Universal Robots PolyScope program: dlo_p0001.urp

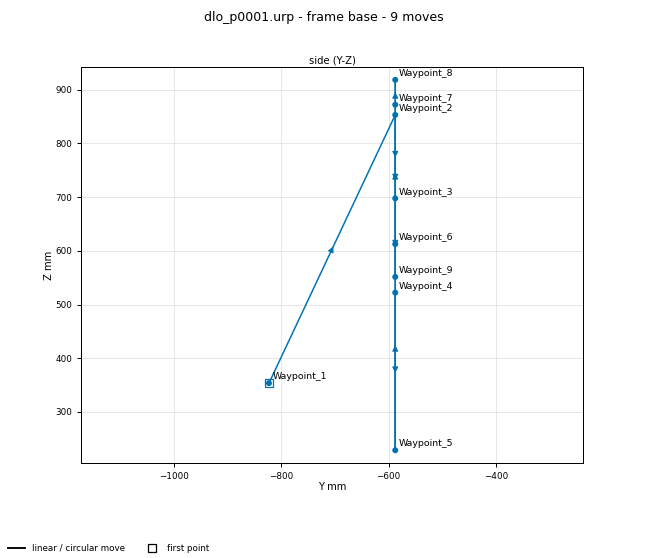
[picture p0: tool path of dlo_p0001.urp in frame base, 9 of 9 moves have a stored position in this frame; points joined in program order, loops and branches not executed]
Program dlo_p0001 (installation=dlo_01 directory=/programs/usbdisk/ur5e createdIn=5.11.4.108353 lastSavedIn=5.11.4.108353 robotSerialNumber=20205500325)
Calibrated DH parameters: a=[0.000117, -0.041718, -0.362867, 0.000002, -0.000002, 0]; d=[0.162762, 132.78066, -173.894578, 41.247059, 0.099793, 0.099638]; alpha=[1.568696, -0.003189, 0.003637, 1.569952, -1.569426, 0]; deltaTheta=[0, -1.472603, 7.364952, 0.390842, 0, 0]
Robot Program (runOnlyOnce=false)
  SetPayload (workpieceName=R2F85_payload)
  MoveJ speed 60 deg/s, acceleration 80 deg/s^2 (useActiveTCP=true) feature=Base
    Waypoint Waypoint_1: TCP in base x=10.232 y=-822.834 z=353.649 mm, rx=0.003 ry=-2.2345 rz=2.1939 rad; joints [76.813, -57.884, 100.068, -221.089, -77.331, -0.468] deg; TCP offset x=0 y=0 z=188 mm, rx=0 ry=0 rz=0 rad
    Popup Message (haltProgram=false message=Bring the DLO near the gripper for gripping, then continue inputType=Text)
    Wait Sleep waitTime=1
    URCap Gripper (Robotiq_Grippers, Robotiq Inc.) dataModel(position=100.0, force=100.0, speed=0.0, positionInDouble=100.0, forceInDouble=100.0, speedInDouble=0.0, slaveIds=[9], blocking=true)
  MoveL speed 250 mm/s, acceleration 1200 mm/s^2 (useActiveTCP=true) feature=Joint_6_name
    Waypoint Waypoint_2: TCP in base x=-0.89 y=-587.732 z=853.044 mm, rx=-0.0177 ry=-2.2261 rz=2.1975 rad; joints [64.46, -101.218, 74.368, -152.362, -65.292, -0.205] deg; feature pose in base x=-0.89 y=-587.732 z=853.044 mm, rx=-0.0177 ry=-2.2261 rz=2.1975 rad
    Waypoint Waypoint_3: TCP in base x=-0.933 y=-587.741 z=697.705 mm, rx=-0.0178 ry=-2.2261 rz=2.1974 rad; joints [64.497, -106.875, 102.164, -174.52, -65.377, -0.152] deg; feature pose in base x=-0.933 y=-587.741 z=697.705 mm, rx=-0.0178 ry=-2.2261 rz=2.1974 rad
    Waypoint Waypoint_4: TCP in base x=-0.931 y=-587.718 z=522.229 mm, rx=-0.0176 ry=-2.2259 rz=2.1975 rad; joints [64.51, -102.812, 125.433, -201.873, -65.499, -0.126] deg; feature pose in base x=-0.931 y=-587.718 z=522.229 mm, rx=-0.0176 ry=-2.2259 rz=2.1975 rad
    Waypoint Waypoint_5: TCP in base x=-0.913 y=-587.718 z=228.776 mm, rx=-0.0178 ry=-2.2261 rz=2.1974 rad; joints [64.493, -57.887, 141.707, -262.996, -65.801, -0.279] deg; feature pose in base x=-0.913 y=-587.718 z=228.776 mm, rx=-0.0178 ry=-2.2261 rz=2.1974 rad
    Waypoint Waypoint_6: TCP in base x=-0.894 y=-587.737 z=612.595 mm, rx=-0.0176 ry=-2.226 rz=2.1975 rad; joints [64.511, -106.524, 114.374, -187.092, -65.43, -0.134] deg; feature pose in base x=-0.894 y=-587.737 z=612.595 mm, rx=-0.0176 ry=-2.226 rz=2.1975 rad
    Waypoint Waypoint_7: TCP in base x=-0.868 y=-587.719 z=872.008 mm, rx=-0.0176 ry=-2.2261 rz=2.1974 rad; joints [64.455, -99.954, 70.248, -149.501, -65.283, -0.217] deg; feature pose in base x=-0.868 y=-587.719 z=872.008 mm, rx=-0.0176 ry=-2.2261 rz=2.1974 rad
    Waypoint Waypoint_8: TCP in base x=-0.882 y=-587.722 z=918.276 mm, rx=-0.0176 ry=-2.226 rz=2.1975 rad; joints [64.438, -96.171, 59.069, -142.1, -65.264, -0.237] deg; feature pose in base x=-0.882 y=-587.722 z=918.276 mm, rx=-0.0176 ry=-2.226 rz=2.1975 rad
    Waypoint Waypoint_9: TCP in base x=-0.931 y=-587.725 z=551.474 mm, rx=-0.0177 ry=-2.226 rz=2.1974 rad; joints [64.511, -104.451, 122.074, -196.868, -65.477, -0.127] deg; feature pose in base x=-0.931 y=-587.725 z=551.474 mm, rx=-0.0177 ry=-2.226 rz=2.1974 rad
